{attribute 'qualified_only'}
{attribute 'strict'}
TYPE Positions :
(
	Position_1 := 4100,
	Position_2 := 12300,
	Position_3 := 20500,
	Position_4 := 28700
);
END_TYPE

(* stored: Version 1.1.0.1, ProductVersion 3.1.4024.11
   DUT Positions: Id {d694dca7-8455-400f-83ea-702652c41a39} *)
